{attribute 'qualified_only'}
{attribute 'strict'}
TYPE StateTr :
(
	Off := 0,
	PowerUp,
	Idle,
	Move2Target,
	Wait,
	Done
);
END_TYPE

(* stored: Version 1.1.0.1, ProductVersion 3.1.4024.3
   DUT StateTr: Id {57c4a080-5a87-4e47-b7cd-a17c062acad1} *)
